FUNCTION_BLOCK Test_WhenReady_Start_SelectsStarting EXTENDS TUnitTestbase
VAR
END_VAR

METHOD  Execute
VAR_INST
    Execution : TExecution;
END_VAR
Test_Started();

Execution.Start();

Assertion.AssertEquals_BOOL(
    Expected := TRUE,
    Actual   := Execution.Starting,
    ObjectName := _TestName,
    VariableName  := 'Execution.Starting');

Test_Finished();
END_METHOD

END_FUNCTION_BLOCK

(* stored: Version 1.1.0.1, ProductVersion 3.1.4024.3
   POU Test_WhenReady_Start_SelectsStarting: Id {02a3c5c8-e774-4d50-adb0-43bf31f75ade}, SpecialFunc None
   Method Execute: Id {c0ea0673-75cd-4bed-bbc1-daf324a7ec7c} *)
